FUNCTION_BLOCK PVDERATOR_NMIN_MEAN (* PV power deration according to N minute running average of grid feed-in power. *)
  (* Standard: 61499-2 *)
  (* Version 0.0, 2017-06-15, Marc Jakobi, HTW Berlin *)
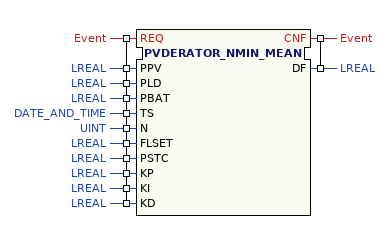
  EVENT_INPUT
    REQ WITH PPV, PLD, PBAT, FLSET, N, TS, PSTC, KP, KI, KD; (* Normal Execution Request *)
  END_EVENT
  EVENT_OUTPUT
    CNF WITH DF; (* Execution Confirmation *)
  END_EVENT
  VAR_INPUT
    PPV : LREAL; (* PV power in W *)
    PLD : LREAL; (* Load in W *)
    PBAT : LREAL; (* Battery power (+charge, -discharge) in W *)
    TS : DATE_AND_TIME; (* Time stamp *)
    N : UINT; (* Time interval of running mean in min *)
    FLSET : LREAL; (* Set limit to N min mean of grid feed-in in kW/kWp *)
    PSTC : LREAL; (* Nominal PV capacity in kWp *)
    KP : LREAL; (* PID proportional coefficient *)
    KI : LREAL := -0.00015313; (* PID integral coefficient *)
    KD : LREAL := 0; (* PID differential coefficient *)
  END_VAR
  VAR_OUTPUT
    DF : LREAL := 1; (* Derating factor *)
  END_VAR
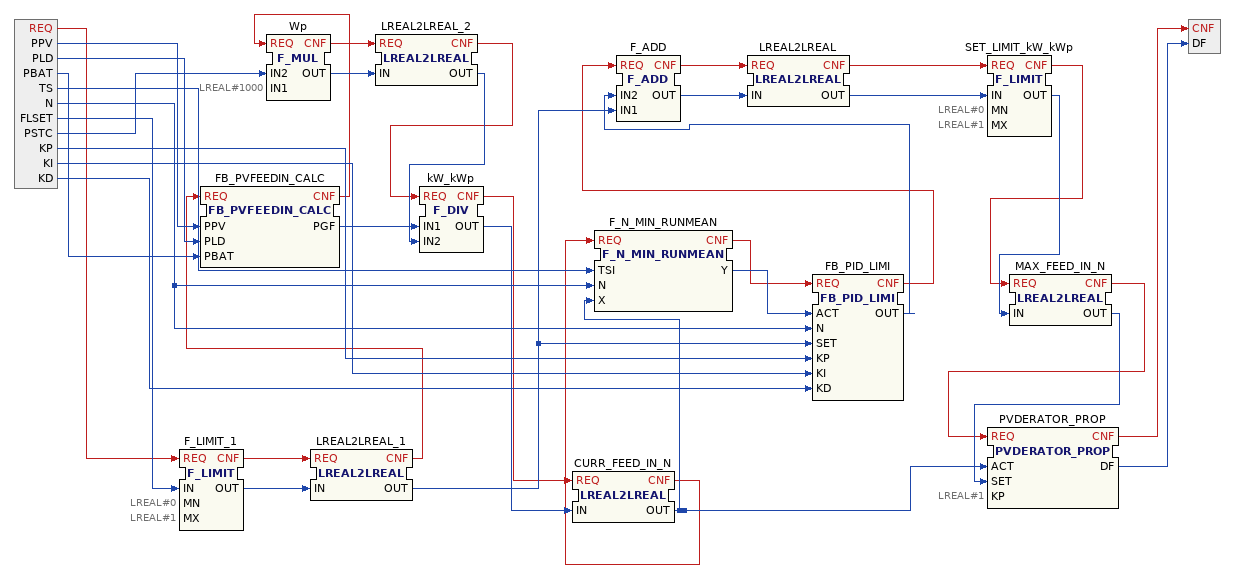
  FBS
    FB_PVFEEDIN_CALC : FB_PVFEEDIN_CALC;
    F_N_MIN_RUNMEAN : F_N_MIN_RUNMEAN;
    FB_PID_LIMI : FB_PID_LIMI;
    F_ADD : F_ADD;
    LREAL2LREAL : LREAL2LREAL;
    SET_LIMIT_kW_kWp : F_LIMIT(MN := LREAL#0, MX := LREAL#1);
    kW_kWp : F_DIV;
    F_LIMIT_1 : F_LIMIT(MN := LREAL#0, MX := LREAL#1);
    LREAL2LREAL_1 : LREAL2LREAL;
    MAX_FEED_IN_N : LREAL2LREAL;
    CURR_FEED_IN_N : LREAL2LREAL;
    PVDERATOR_PROP : PVDERATOR_PROP(KP := LREAL#1);
    Wp : F_MUL(IN1 := LREAL#1000);
    LREAL2LREAL_2 : LREAL2LREAL;
  END_FBS
  EVENT_CONNECTIONS
    F_ADD.CNF TO LREAL2LREAL.REQ;
    LREAL2LREAL.CNF TO SET_LIMIT_kW_kWp.REQ;
    REQ TO F_LIMIT_1.REQ;
    FB_PID_LIMI.CNF TO F_ADD.REQ;
    F_LIMIT_1.CNF TO LREAL2LREAL_1.REQ;
    LREAL2LREAL_1.CNF TO FB_PVFEEDIN_CALC.REQ;
    SET_LIMIT_kW_kWp.CNF TO MAX_FEED_IN_N.REQ;
    kW_kWp.CNF TO CURR_FEED_IN_N.REQ;
    CURR_FEED_IN_N.CNF TO F_N_MIN_RUNMEAN.REQ;
    F_N_MIN_RUNMEAN.CNF TO FB_PID_LIMI.REQ;
    MAX_FEED_IN_N.CNF TO PVDERATOR_PROP.REQ;
    PVDERATOR_PROP.CNF TO CNF;
    FB_PVFEEDIN_CALC.CNF TO Wp.REQ;
    Wp.CNF TO LREAL2LREAL_2.REQ;
    LREAL2LREAL_2.CNF TO kW_kWp.REQ;
  END_CONNECTIONS
  DATA_CONNECTIONS
    PPV TO FB_PVFEEDIN_CALC.PPV;
    PLD TO FB_PVFEEDIN_CALC.PLD;
    PBAT TO FB_PVFEEDIN_CALC.PBAT;
    TS TO F_N_MIN_RUNMEAN.TSI;
    N TO F_N_MIN_RUNMEAN.N;
    F_N_MIN_RUNMEAN.Y TO FB_PID_LIMI.ACT;
    N TO FB_PID_LIMI.N;
    FB_PID_LIMI.OUT TO F_ADD.IN2;
    F_ADD.OUT TO LREAL2LREAL.IN;
    LREAL2LREAL.OUT TO SET_LIMIT_kW_kWp.IN;
    FB_PVFEEDIN_CALC.PGF TO kW_kWp.IN1;
    FLSET TO F_LIMIT_1.IN;
    LREAL2LREAL_1.OUT TO F_ADD.IN1;
    F_LIMIT_1.OUT TO LREAL2LREAL_1.IN;
    LREAL2LREAL_1.OUT TO FB_PID_LIMI.SET;
    SET_LIMIT_kW_kWp.OUT TO MAX_FEED_IN_N.IN;
    kW_kWp.OUT TO CURR_FEED_IN_N.IN;
    CURR_FEED_IN_N.OUT TO F_N_MIN_RUNMEAN.X;
    CURR_FEED_IN_N.OUT TO PVDERATOR_PROP.ACT;
    MAX_FEED_IN_N.OUT TO PVDERATOR_PROP.SET;
    PVDERATOR_PROP.DF TO DF;
    PSTC TO Wp.IN2;
    Wp.OUT TO LREAL2LREAL_2.IN;
    LREAL2LREAL_2.OUT TO kW_kWp.IN2;
    KP TO FB_PID_LIMI.KP;
    KI TO FB_PID_LIMI.KI;
    KD TO FB_PID_LIMI.KD;
  END_CONNECTIONS
END_FUNCTION_BLOCK
